INTERFACE I_HostContent

PROPERTY PUBLIC Contents : I_Contents
GET
END_GET
END_PROPERTY

END_INTERFACE

(* stored: Version 1.1.0.1, ProductVersion 3.1.4024.12
   Itf I_HostContent: Id {e1e0eb08-bfd1-4547-a6bc-473321063a08}
   Property Contents: Id {b49ca806-3c29-4d74-a1af-1efc03a7ce91}
   Get Get: Id {88e896f6-b846-463e-9fb3-0f24acf0c655} *)
